FUNCTION_BLOCK EL1809
VAR
	DI_ESR1_tmp : DIChannel;
END_VAR

END_FUNCTION_BLOCK

(* stored: Version 1.1.0.1, ProductVersion 3.1.4024.6
   POU EL1809: Id {2d9d8afb-39a4-4fda-a15a-2bc58d6817d2}, SpecialFunc None *)
